FUNCTION_BLOCK MC_HomeAxis
VAR_INPUT
	xExecute		: BOOL;
	xReset			: BOOL;
END_VAR

VAR
	eStates 		: E_HomingSteps :=E_HomingSteps.IDLE;
	rtHomeStart		: R_TRIG;
	rtHomeReset		: R_TRIG;
	ton_delay		: TON;
	bError			: BOOL;	
END_VAR
VAR_IN_OUT
	InOut		: ST_MotionAxis_MC;
END_VAR
VAR_OUTPUT
	xRedy		: BOOL;
	xBusy		: BOOL;
	xDone		: BOOL;
	xError		: BOOL;
END_VAR

rtHomeStart(CLK:=xExecute);
rtHomeReset(CLK:=xReset);
ton_delay(PT:= T#2S);

IF rtHomeStart.Q THEN
	eStates := E_HomingSteps.START;
END_IF
IF rtHomeReset.Q THEN
	eStates := E_HomingSteps.IDLE;
END_IF
IF InOut.mcStop.Execute THEN
	eStates := E_HomingSteps.ERROR;
END_IF
CASE eStates OF
		E_HomingSteps.IDLE:// WAIT FOR REQUEST	
	//Wait for Reset
		IF rtHomeReset.Q THEN
			InOut.mcReset.Execute := TRUE;
			InOut.mcJog.JogForward :=FALSE;
			InOut.mcJog.JogBackwards :=FALSE;
			xExecute := FALSE;
			bError := FALSE;
		END_IF	
		InOut.xHoming	:= FALSE;
	E_HomingSteps.INIT:		
		;

	E_HomingSteps.START:
			ton_delay.IN	:= FALSE;
			InOut.xHoming	:= TRUE;
			InOut.rVeloPers :=30;
			IF InOut.bdirFW THEN//first direction
				eStates := E_HomingSteps.JOG_FW;	
			ELSE
				eStates := E_HomingSteps.JOG_BW;	
			END_IF
///////////////////////////////////////////////////////////////////////////	
	E_HomingSteps.JOG_FW:
		IF InOut.bPosSen THEN
			InOut.mcJog.JogForward :=TRUE;			
		ELSE
			InOut.mcJog.JogForward :=FALSE;
			eStates := E_HomingSteps.JOG_BW_DOG;			
		END_IF
	E_HomingSteps.JOG_BW_DOG:
		IF InOut.bPositionSensor THEN
			InOut.mcJog.JogBackwards :=FALSE;
			eStates := E_HomingSteps.FW_DOG_OFF;			
		ELSE
			InOut.mcJog.JogBackwards :=TRUE;
		END_IF	
	E_HomingSteps.FW_DOG_OFF:	
		IF InOut.bPositionSensor THEN
			InOut.mcJog.JogForward := TRUE;
			InOut.rVeloPers	:=	5;						
		ELSE
			InOut.mcJog.JogForward := FALSE;
			eStates := E_HomingSteps.BW_DOG_ON;
		END_IF		
	E_HomingSteps.BW_DOG_ON:
		IF InOut.bPositionSensor THEN
			InOut.mcJog.JogBackwards := FALSE;
			eStates := E_HomingSteps.WAIT;					
		ELSE
			InOut.rVeloPers	:=	2;		
			InOut.mcJog.JogBackwards := TRUE;		
		END_IF		
///////////////////////////////////////////////////////////////////////////	
	E_HomingSteps.JOG_BW:
		IF InOut.bNegSen THEN
			InOut.mcJog.JogBackwards :=TRUE;			
		ELSE
			InOut.mcJog.JogBackwards :=FALSE;
			eStates := E_HomingSteps.JOG_FW_DOG;	
		END_IF
	E_HomingSteps.JOG_FW_DOG:
		IF InOut.bPositionSensor THEN
			InOut.mcJog.JogForward :=FALSE;
			eStates := E_HomingSteps.BW_DOG_OFF;				
		ELSE
			InOut.mcJog.JogForward :=TRUE;
		END_IF	
	E_HomingSteps.BW_DOG_OFF:	
		IF InOut.bPositionSensor THEN
			InOut.mcJog.JogBackwards := TRUE;
			InOut.rVeloPers	:=	5;						
		ELSE
			InOut.mcJog.JogBackwards := FALSE;
			eStates := E_HomingSteps.FW_DOG_ON;
		END_IF		
	E_HomingSteps.FW_DOG_ON:
		IF InOut.bPositionSensor THEN
			InOut.mcJog.JogForward := FALSE;
			eStates := E_HomingSteps.WAIT;					
		ELSE
			InOut.rVeloPers	:=	2;		
			InOut.mcJog.JogForward := TRUE;		
		END_IF		
///////////////////////////////////////////////////////////////////////////
	E_HomingSteps.WAIT:
		ton_delay.IN	:= TRUE;
		IF ton_delay.Q THEN
			eStates := E_HomingSteps.MCHOME;	
		END_IF
	E_HomingSteps.MCHOME:
		IF InOut.mcReadStatus.StandStill THEN
			InOut.mcHome.Execute := TRUE;	
		END_IF
		IF NOT InOut.mcHome.Busy AND InOut.mcHome.Done THEN
			InOut.mcHome.Execute := FALSE;
			eStates := E_HomingSteps.DONE;	
		END_IF		
	E_HomingSteps.DONE:	
		InOut.xHoming	:= FALSE;
		InOut.xHomingDone	:= TRUE;
		InOut.rVeloPers	:=	10;	
		eStates := E_HomingSteps.IDLE;	
		
	E_HomingSteps.ERROR:	
		InOut.mcJog.JogForward :=FALSE;
		InOut.mcJog.JogBackwards :=FALSE;
		IF InOut.mcReadStatus.Error THEN
			InOut.xHomingDone	:= FALSE;
		END_IF		
		eStates := E_HomingSteps.IDLE;	
		
END_CASE

xRedy		:= (eStates = E_HomingSteps.IDLE);
xBusy		:= (eStates > E_HomingSteps.IDLE AND eStates < E_HomingSteps.DONE);
xDone		:= (eStates = E_HomingSteps.DONE );
xError		:= (eStates = E_HomingSteps.ERROR);

END_FUNCTION_BLOCK

(* stored: Version 1.1.0.1, ProductVersion 3.1.4024.12
   POU MC_HomeAxis: Id {994399f9-7878-4425-887e-8af0d446f64c}, SpecialFunc None *)
